Staubli VAL3: create_plane.pgx

public program create_plane(point x_pOrigin, point x_pPointX, point x_pPointY)
begin
  //
  // build the plane
  //
  // Origin
  if setFrame(x_pOrigin,x_pPointX,x_pPointY,fPlane)==0
    bCreate_plane=true
  else
    bCreate_plane=false
  endIf
end
